// TIA Portal V18 export
FUNCTION "ST10_PartData" : Void   // FC1500, SCL
{ S7_Optimized_Access := 'TRUE' }
VERSION : 0.1
// stored: AutoNumber true, IsIECCheckEnabled false, SetENOAutomatically false, UDAEnableTagReadback false
   VAR_INPUT
      iSysMode : "RCS_SysComInterface_V1";
   END_VAR
   VAR_TEMP
      idex : Int;
   END_VAR
BEGIN
END_FUNCTION
